PROGRAM MAIN
VAR
	
END_VAR


SignalHandler();
	
//======================Handl the signal from UI=================== 
	LinkUI();
//======================Handl the signal from UI=================== 



//======================Handl the signal from Hardware===================
	LinkHWIO();
//======================Handl the signal from Hardware===================





//====================handle the lights rolling======================
	LampControl();
//====================handle the lights rolling======================

//=========Machine mode selecion================
	ModeManger();
//=========Machine mode selecion================

END_PROGRAM

(* stored: Version 1.1.0.1, ProductVersion 3.1.4022.16
   POU MAIN: Id {3842b7b5-2d54-412a-975a-36a7ea8a0c51}, SpecialFunc None *)
